FUNCTION_BLOCK PUBLIC FB_LampSetDirect EXTENDS FB_Lamp
VAR
	nLightLevel			: BYTE(0..100);
END_VAR

// Reduces the control value by 5 in the range of 10 to 100.
METHOD PUBLIC DimDown
IF (nLightLevel >= 15) THEN
	SetLightLevel(nLightLevel - 5);
END_IF
END_METHOD

// Increments the control value by 5 in the range of 10 to 100.
METHOD PUBLIC DimUp
IF (nLightLevel <= 95) THEN
	SetLightLevel(nLightLevel + 5);
END_IF
END_METHOD

// Sets the control value to 0.
METHOD PUBLIC Off
SetLightLevel(0);
END_METHOD

// Sets the control value to 100.
METHOD PUBLIC On
SetLightLevel(100);
END_METHOD

// Sets the control value to a value between 0 and 100.
METHOD PUBLIC SetLightLevel
VAR_INPUT
	nNewLightLevel		: BYTE(0..100);
END_VAR
nLightLevel := nNewLightLevel;
IF (_ipObserver <> 0) THEN
	_ipObserver.Update(nLightLevel);
END_IF
END_METHOD

END_FUNCTION_BLOCK

(* stored: Version 1.1.0.1, ProductVersion 3.1.4024.9
   POU FB_LampSetDirect: Id {c9363aa1-33e3-41da-adea-7faeb59d6855}, SpecialFunc None
   Method DimDown: Id {b90d3b74-1a90-4f15-84df-bd103eb2839f}
   Method DimUp: Id {14eaeaf5-74a2-48eb-83f1-083b8b2dce0e}
   Method Off: Id {28372a2b-69a1-43d3-97df-f71c4a0264b6}
   Method On: Id {c86e14d4-f798-4427-9c52-89a5594d2119}
   Method SetLightLevel: Id {4b6fea93-5fee-4ee1-8a77-261782e46dcf} *)
